FUNCTION TryConvert_USINT_TO_SINT : BOOL
VAR_INPUT
	in : USINT;
	out : REFERENCE TO SINT;
END_VAR

IF in > DatatypeLimits.MAX_VALUE_OF_USINT_WHICH_CAN_BE_HELD_IN_A_SINT THEN
	RETURN;
END_IF

out := USINT_TO_SINT(in);
TryConvert_USINT_TO_SINT := TRUE;

END_FUNCTION

(* stored: Version 1.1.0.1, ProductVersion 3.1.4024.12
   POU TryConvert_USINT_TO_SINT: Id {ad4ac2be-5086-43d3-9ba1-79a28bffd79e}, SpecialFunc None *)
